(* PLC project Senza_nome, Sconosciuto Senza_nome 1 *)
(* stored: creationDateTime 2026-08-25T12:02:26, modificationDateTime 2026-08-25T12:32:47 *)

PROGRAM program0
  VAR
    P1 : BOOL;
    P2 : BOOL;
    P3 : BOOL;
    P4 : BOOL;
    P5 : BOOL;
    P6 : BOOL;
    P7 : BOOL;
    LED1 : BOOL;
    LED2 : BOOL;
    LED3 : BOOL;
    LED4 : BOOL;
  END_VAR

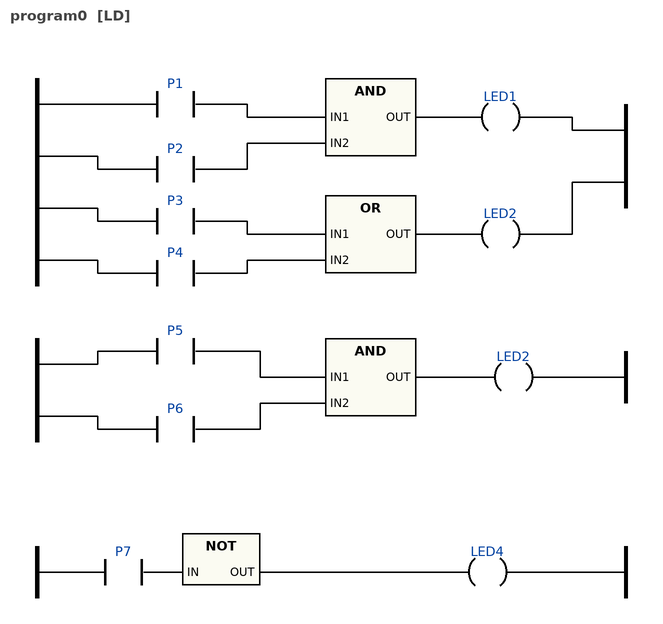
(* LD diagram, written out as Structured Text *)
LED1 := P1 AND P2;
LED2 := P3 OR P4;
LED2 := P5 AND P6;
LED4 := NOT P7;
END_PROGRAM

CONFIGURATION Config0
  RESOURCE Res0 ON PLC
    TASK task0(INTERVAL := T#20ms, PRIORITY := 0);
    PROGRAM instance0 WITH task0 : program0;
  END_RESOURCE
END_CONFIGURATION
